Staubli VAL3: refresh.pgx

program refresh()
// // page refresh
begin
  if (nKey>=270 and nKey<=278) or use:bUseRefresh
    cls()
    call refreshStatic()
    call buildList()
    call refreshDynamic()
  else
    //refresh the Dynamic message
    if (clock()-nRefresh>nTime)
      call refreshDynamic()
    endIf
  endIf
  delay(0.1)
end
